FUNCTION_BLOCK RemoveAllMoverFromGroup IMPLEMENTS ITask
VAR_INPUT
END_VAR
VAR_OUTPUT
END_VAR
VAR
	RemoveAllFromGrp			: MC_UngroupAllAxes;
	_caGroup			: ICollisionGroup;
	State: INT;
	_removeAllMovers : BOOL;
	_busy : BOOL;
	_error : BOOL;
	_done : BOOL;
	_moverNumber : INT;
	_errorId: UDINT;
END_VAR

CASE State OF
	0:
		IF _removeAllMovers THEN
			_done := FALSE;
			_error := FALSE;
			_busy := TRUE;
			RemoveAllFromGrp.Execute := TRUE;
			IF RemoveAllFromGrp.Busy THEN
				_removeAllMovers := FALSE;
				State := 10;
			END_IF
		END_IF
		
	10:
		IF NOT RemoveAllFromGrp.Busy THEN
			IF RemoveAllFromGrp.Done THEN
				_done := TRUE;
			ELSIF RemoveAllFromGrp.Error THEN
				_error := TRUE;
				_errorId := RemoveAllFromGrp.ErrorId;
			END_IF
			_busy := FALSE;
			RemoveAllFromGrp.Execute := false;
			State := 0;
		END_IF
END_CASE


RemoveAllFromGrp(AxesGroup := _caGroup.GroupRef);

METHOD Abort : BOOL
RemoveAllFromGrp.Execute := FALSE;
Abort := true;
State := 0;
END_METHOD


PROPERTY Busy : BOOL
GET
Busy := _busy;
END_GET
END_PROPERTY


PROPERTY Done : BOOL
GET
Done := _done;
END_GET
END_PROPERTY


PROPERTY Error : BOOL
GET
Error := _error;
END_GET
END_PROPERTY

METHOD FB_init : BOOL
VAR_INPUT
	bInitRetains : BOOL; // if TRUE, the retain variables are initialized (warm start / cold start)
	bInCopyCode : BOOL;  // if TRUE, the instance afterwards gets moved into the copy code (online change)
	CAGroup : ICollisionGroup;	
END_VAR
_caGroup := CAGroup;
END_METHOD

METHOD RemoveAllMover : BOOL
RemoveAllMover := _removeAllMovers := true;
END_METHOD

END_FUNCTION_BLOCK

(* stored: Version 1.1.0.1, ProductVersion 3.1.4024.11
   POU RemoveAllMoverFromGroup: Id {047a0fff-03f1-4967-ab6d-21073bd96b33}, SpecialFunc None
   Method Abort: Id {5bfcf5d7-ad93-4041-89c5-a1c0c5514d79}
   Property Busy: Id {0da215af-4e15-45ae-b6df-6bfb3fbd8c09}
   Get Get: Id {4bcf1385-240e-4de2-8c06-7ea23165eaa9}
   Property Done: Id {d30b6d2d-8329-4441-bd1d-4ea3064e7851}
   Get Get: Id {a0b4ac09-0b1c-49ac-8d09-bc0314287f1f}
   Property Error: Id {2429d49d-82c4-46cf-9cd6-0f8f7f8528d8}
   Get Get: Id {58129a3f-70ec-4d42-8026-1a44d11299d5}
   Method FB_init: Id {21970abf-5278-4aab-8753-fe6ec776ee38}
   Method RemoveAllMover: Id {1e71b9a7-d764-4dd3-a760-276d6f124ab0} *)
